{attribute 'GeneratedUsingTerminal: KL6551'}
{attribute addProperty BoxType "KL6551"}
{attribute addProperty Id "Parameter_StatusAT %I*UINT0Input_Data_1AT %I*USINT0Input_Data_2AT %I*USINT0Input_Data_3AT %I*USINT0Input_Data_4AT %I*USINT0Input_Data_5AT %I*USINT0Input_Data_6AT %I*USINT0Input_Data_7AT %I*USINT0Input_Data_8AT %I*USINT0Input_Data_9AT %I*USINT0Input_Data_10AT %I*USINT0Parameter_ControlAT %Q*UINT0Output_Data_1AT %Q*USINT0Output_Data_2AT %Q*USINT0Output_Data_3AT %Q*USINT0Output_Data_4AT %Q*USINT0Output_Data_5AT %Q*USINT0Output_Data_6AT %Q*USINT0Output_Data_7AT %Q*USINT0Output_Data_8AT %Q*USINT0Output_Data_9AT %Q*USINT0Output_Data_10AT %Q*USINT0"}
{attribute addProperty CRC "1764871259"}
{attribute addProperty Size "0"}
TYPE Channel_6931CC5B :
STRUCT
	{attribute addProperty Name "Parameter_Status"}
	Parameter_Status AT %I* : UINT;
	{attribute addProperty Name "Input_Data_1"}
	Input_Data_1 AT %I* : USINT;
	{attribute addProperty Name "Input_Data_2"}
	Input_Data_2 AT %I* : USINT;
	{attribute addProperty Name "Input_Data_3"}
	Input_Data_3 AT %I* : USINT;
	{attribute addProperty Name "Input_Data_4"}
	Input_Data_4 AT %I* : USINT;
	{attribute addProperty Name "Input_Data_5"}
	Input_Data_5 AT %I* : USINT;
	{attribute addProperty Name "Input_Data_6"}
	Input_Data_6 AT %I* : USINT;
	{attribute addProperty Name "Input_Data_7"}
	Input_Data_7 AT %I* : USINT;
	{attribute addProperty Name "Input_Data_8"}
	Input_Data_8 AT %I* : USINT;
	{attribute addProperty Name "Input_Data_9"}
	Input_Data_9 AT %I* : USINT;
	{attribute addProperty Name "Input_Data_10"}
	Input_Data_10 AT %I* : USINT;
	{attribute addProperty Name "Parameter_Control"}
	Parameter_Control AT %Q* : UINT;
	{attribute addProperty Name "Output_Data_1"}
	Output_Data_1 AT %Q* : USINT;
	{attribute addProperty Name "Output_Data_2"}
	Output_Data_2 AT %Q* : USINT;
	{attribute addProperty Name "Output_Data_3"}
	Output_Data_3 AT %Q* : USINT;
	{attribute addProperty Name "Output_Data_4"}
	Output_Data_4 AT %Q* : USINT;
	{attribute addProperty Name "Output_Data_5"}
	Output_Data_5 AT %Q* : USINT;
	{attribute addProperty Name "Output_Data_6"}
	Output_Data_6 AT %Q* : USINT;
	{attribute addProperty Name "Output_Data_7"}
	Output_Data_7 AT %Q* : USINT;
	{attribute addProperty Name "Output_Data_8"}
	Output_Data_8 AT %Q* : USINT;
	{attribute addProperty Name "Output_Data_9"}
	Output_Data_9 AT %Q* : USINT;
	{attribute addProperty Name "Output_Data_10"}
	Output_Data_10 AT %Q* : USINT;
END_STRUCT
END_TYPE

(* stored: Version 1.2.0.0, ProductVersion 3.1.4024.9
   DUT Channel_6931CC5B: Id {896ac01d-f69c-4f1f-b1d7-9aedd26b1026} *)
